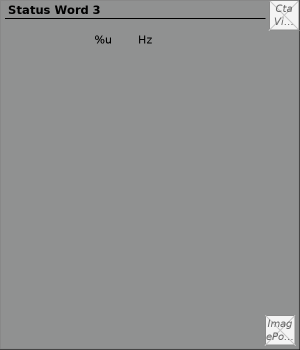
VISUALIZATION VERDICHTER_BUS_SW3_Detail  // 300x350
VAR_IN_OUT
    wDetail             :   WORD;
END_VAR
VAR_INPUT	
    ITF_VERDICHTERIN       :   ITF_VERDICHTER;
END_VAR
VAR_IN_OUT
    xShow               :   BOOL;
END_VAR
    Rectangle (0,0 300x350)
    Image (269,0 30x30), image: CtaVisSymbols.ImagePool.close_solo_black
        OnMouseClick: execute { xShow := FALSE; ITF_VERDICHTERIN.proModbusTest := FALSE; }
    Label (5,0 150x20), "Status Word 3"
    Image (265,315 30x30), invisible if: ITF_VERDICHTERIn.proModbusTest, image: ImagePool.front_hand_FILL0_wght400_GRAD0_opsz48
        OnMouseClick: execute { ITF_VERDICHTERIN.proModbusTest := TRUE; }
    Image (265,315 30x30), invisible if: NOT ITF_VERDICHTERIN.proModbusTest, image: ImagePool.front_hand_FILL0_wght400_GRAD0_opsz48Yellow
        OnMouseClick: execute { ITF_VERDICHTERIN.proModbusTest := False; }
    Label (135,30 120x20), "Hz"
    Textfield (5,30 110x20), "%u", text variable: wDetail, input disabled if: NOT ITF_VERDICHTERIn.proModbusTest
        OnMouseClick: write the text variable via InputWithLimits, min 0, max 100
    Textfield (5,30 110x20), "%u", text variable: wDetail, invisible if: ITF_VERDICHTERIN.proModbusTest
    Line (5,18) (265,18)
END_VISUALIZATION

// 40 Visualizations/ICON/VERDICHTER_BASE/VALUE/ValueDwnUp
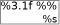
VISUALIZATION ValueDwnUp  // 60x25
VAR_INPUT
    ITF_VERDICHTER_IN   :   ITF_VERDICHTER;	
END_VAR
VAR_INPUT CONSTANT
    uiTextAusrichtung   : UINT := 4;    // 0 = Oben links | 1 = Horizontal zentriert | 2 = Rechts | 4 = Vertikal zentriert | 8 = Unten
END_VAR
    Textfield (0,13 60x12), "%s", text variable: ITF_VERDICHTER_IN.proGetBMK, invisible if: ITF_VERDICHTER_IN.proNoBmkInList
        p3718999670: uiTextAusrichtung
    Textfield (0,0 60x12), "%3.1f %%", text variable: ITF_VERDICHTER_IN.proLeistung, invisible if: NOT ITF_VERDICHTER_IN.proIsRegulatet
        p3718999670: uiTextAusrichtung
END_VISUALIZATION

(* text list Error (id | default | de | en | fr | it)
  0 | keine Meldung Anstehend | Keine Meldung Anstehend | No message pending | Aucun message en attente | Nessun messaggio in sospeso
  1 | keine Betriebsrückmeldung | Keine Betriebsrückmeldung | No operational feedback | Aucune rétroaction opérationnelle | Nessun feedback operativo
  2 | Alarmkontakt Anstehend | Alarmkontakt Anstehend | Error contact pending | Contact d'alarme en attente | Contatto di allarme in sospeso
  3 | Leitungsschutzschalter ausfall | Leitungsschutzschalter ausfall | Circuit breaker failure | Défaillance du disjoncteur | Guasto dell'interruttore
  4 | Motorschutzschalter ausfall | Motorschutzschalter ausfall | Motor protection switch failure | Défaillance de l'interrupteur de protection du moteur | Guasto al salvamotore
  5 | Konfigurationsfehler speichern fehlgeschlagen reboot | Konfigurationsfehler speichern fehlgeschlagen reboot | Failed to save configuration error reboot | Impossible d'enregistrer l'erreur de configuration reboot | Impossibile salvare l'errore di configurazione reboot
   |  |  |  |  |  *)

(* text list Info (id | default | de | en | fr | it)
  0 | keine Meldung Anstehend | keine Meldung Anstehend | no message pending | aucun message en attente | nessun messaggio in sospeso
   |  |  |  |  |  *)

(* text list Warnung (id | default | de | en | fr | it)
  0 | Keine Meldung Anstehend | Keine Meldung Anstehend | No message pending | Aucun message en attente | Nessun messaggio in sospeso
  4 | Wahlschalter Hand, Ein | Wahlschalter Hand, Ein | Selector switch hand on | Commutateur de sélection a main, Allumé | Selettore a mano, acceso
  3 | Wahlschalter Hand, Aus | Wahlschalter Hand, Aus | Selector switch hand off | Commutateur de sélection a main, Éteint | Selettore a mano, spento
  2 | Revisionsschalter Ausgeschalten | Revisionsschalter Ausgeschalten | Revision switch off | Commutateur révision Désactiver | Interruttore di revisione disattivato
  1 | Sicherheits Stopp | Sicherheits Stopp | Safety stop | Arrêt de sécurité | Sosta di sicurezza
  5 | Handmodul aktiv | Handmodul aktiv | Hand module active | Module manuel actif | Modulo manuale attivo
   |  |  |  |  |  *)
